{attribute 'qualified_only'}
VAR_GLOBAL CONSTANT
	MAX_TASK_NUM : UINT := 10; // Number of max jobs in job container object.
	MAX_STRING_LENGTH : UDINT := 255; // Max string length of task name.
END_VAR

(* stored: Version 1.1.0.1, ProductVersion 3.1.4024.12
   GVL ParamFuturesLib: Id {8c42569b-1214-437d-89e7-2037e9eec4b9}, ParameterList True *)
